TEXTLIST MessageList
  0 = ' '
  1 = 'MENSAGEM DE ADVERTENCIA 01'
  2 = 'MENSAGEM DE ADVERTENCIA 02'
  3 = 'MENSAGEM DE ADVERTENCIA 03'
  4 = 'MENSAGEM DE ADVERTENCIA 04'
  5 = 'MENSAGEM DE ADVERTENCIA 05'
  6 = 'MENSAGEM DE ADVERTENCIA 06'
  7 = 'MENSAGEM DE ADVERTENCIA 07'
  8 = 'MENSAGEM DE ADVERTENCIA 08'
  9 = 'MENSAGEM DE ADVERTENCIA 09'
  10 = 'MENSAGEM DE ADVERTENCIA 10'
  11 = 'MENSAGEM DE ADVERTENCIA ...'
  12 = 'MENSAGEM DE ADVERTENCIA ...'
  13 = 'MENSAGEM DE ADVERTENCIA ...'
  14 = 'MENSAGEM DE ADVERTENCIA ...'
  15 = 'MENSAGEM DE ADVERTENCIA ...'
  99 = 'MENSAGEM DE ADVERTENCIA 99'
  101 = 'MENSAGEM DE ALARME 01'
  102 = 'MENSAGEM DE ALARME 02'
  103 = 'MENSAGEM DE ALARME 03'
  104 = 'MENSAGEM DE ALARME 04'
  105 = 'MENSAGEM DE ALARME 05'
  106 = 'MENSAGEM DE ALARME 06'
  107 = 'MENSAGEM DE ALARME 07'
  108 = 'MENSAGEM DE ALARME 08'
  109 = 'MENSAGEM DE ALARME 09'
  110 = 'MENSAGEM DE ALARME 10'
  111 = 'MENSAGEM DE ALARME ...'
  299 = 'MENSAGEM DE ALARME 299'
   = ''
END_TEXTLIST

(* stored: Version 1.1.0.1, ProductVersion 3.1.4024.12
   TextList MessageList: Id {c034b06b-6010-40a3-8a2a-dc1da4b4d518} *)
